{attribute 'GeneratedUsingTerminal: EP7041-0002-0016'}
{attribute addProperty BoxType "EP7041-0002-0016"}
{attribute addProperty Id "AdsAddrAT %I*AMSADDR8Chn0AT %I*USINT1StateAT %I*UINT2"}
{attribute addProperty CRC "2381635781"}
{attribute addProperty Size "11"}
TYPE InfoData_8DF4E0C5 :
STRUCT
	{attribute addProperty Name "AdsAddr"}
	AdsAddr AT %I* : AMSADDR;
	{attribute addProperty Name "Chn0"}
	Chn0 AT %I* : USINT;
	{attribute addProperty Name "State"}
	State AT %I* : UINT;
END_STRUCT
END_TYPE

(* stored: Version 1.2.0.0, ProductVersion 3.1.4024.9
   DUT InfoData_8DF4E0C5: Id {bf9e7930-3e7d-46df-8cde-3a820fbd7332} *)
